// TIA Portal V17 export
// export: Created 2024-09-15T12:30:20.7468626Z, ExportSetting WithDefaults, DisplayName Totally Integrated Automation Portal, DisplayVersion V17, DisplayName TIA Portal Openness, DisplayVersion V17, DisplayName TIA Portal Version Control Interface, DisplayVersion V17, DisplayName STEP 7 Professional, DisplayVersion V17, DisplayName STEP 7 Safety, DisplayVersion V17, DisplayName WinCC Professional, DisplayVersion V17
VAR_GLOBAL   // PLC tag table "VGR - Vacuum Gripper Robot"
   IX_VGR_RefSwitchVerticalAxis_I1 AT %I1.6 : Bool;   // VGR - I1 = Reference switch vertical axis   {ExternalAccessible false, ExternalVisible false, ExternalWritable false}
   IX_VGR_RefSwitchHorizontalAxis_I2 AT %I3.6 : Bool;   // VGR - I2 = Reference switch horizontal axis   {ExternalAccessible false, ExternalVisible false, ExternalWritable false}
   IX_VGR_RefSwitchRotate_I3 AT %I3.7 : Bool;   // VGR - I3 = Reference switch rotate   {ExternalAccessible false, ExternalVisible false, ExternalWritable false}
   IX_VGR_EncoderVerticalAxisImp1_B1 AT %I6.0 : Bool;   // VGR - B1 = Encoder vertical axis imulse 1   {ExternalAccessible false, ExternalVisible false, ExternalWritable false}
   IX_VGR_EncoderVerticalAxisImp2_B2 AT %I6.4 : Bool;   // VGR - B2 = Encoder vertical axis imulse 2   {ExternalAccessible false, ExternalVisible false, ExternalWritable false}
   IX_VGR_EncoderHorizontalAxisImp1_B3 AT %I6.1 : Bool;   // VGR - B3 = Encoder horizontal axis imulse 1   {ExternalAccessible false, ExternalVisible false, ExternalWritable false}
   IX_VGR_EncoderHorizontalAxisImp2_B4 AT %I6.5 : Bool;   // VGR - B4 = Encoder horizontal axis imulse 2   {ExternalAccessible false, ExternalVisible false, ExternalWritable false}
   IX_VGR_EncoderRotateImp1_B5 AT %I6.2 : Bool;   // VGR - B5 = Encoder rotate impulse 1   {ExternalAccessible false, ExternalVisible false, ExternalWritable false}
   IX_VGR_EncoderRotateImp2_B6 AT %I6.6 : Bool;   // VGR - B6 = Encoder rotate impulse 2   {ExternalAccessible false, ExternalVisible false, ExternalWritable false}
   QX_VGR_M1_VerticalAxisUp_Q1 AT %Q2.0 : Bool;   // VGR - Q1 = Motor M1 vertical axis up   {ExternalAccessible false, ExternalVisible false, ExternalWritable false}
   QX_VGR_M1_VerticalAxisDown_Q2 AT %Q2.1 : Bool;   // VGR - Q2 = Motor M1 vertical axis down   {ExternalAccessible false, ExternalVisible false, ExternalWritable false}
   QX_VGR_M2_HorizontalAxisBackward_Q3 AT %Q2.2 : Bool;   // VGR - Q3 = Motor M2 horizontal axis backward   {ExternalAccessible false, ExternalVisible false, ExternalWritable false}
   QX_VGR_M2_HorizontalAxisForward_Q4 AT %Q2.3 : Bool;   // VGR - Q4 = Motor M2 horizontal axis forward   {ExternalAccessible false, ExternalVisible false, ExternalWritable false}
   QX_VGR_M3_RotateClockwise_Q5 AT %Q2.4 : Bool;   // VGR - Q5 = Motor M3 rotate clockwise   {ExternalAccessible false, ExternalVisible false, ExternalWritable false}
   QX_VGR_M3_RotateCounterclockwise_Q6 AT %Q2.5 : Bool;   // VGR - Q6 = Motor M3 rotate counterclockwise   {ExternalAccessible false, ExternalVisible false, ExternalWritable false}
   QX_VGR_Compressor_Q7 AT %Q2.6 : Bool;   // VGR - Q7 = Compressor   {ExternalAccessible false, ExternalVisible false, ExternalWritable false}
   QX_VGR_ValveVacuum_Q8 AT %Q2.7 : Bool;   // VGR - Q8 = Valve vacuum   {ExternalAccessible false, ExternalVisible false, ExternalWritable false}
   QW_VGR_PWM_Vertical_M1 AT %QW15 : Int;   // VGR = PWM Motor M1 vertical axis   {ExternalAccessible false, ExternalVisible false, ExternalWritable false}
   QW_VGR_PWM_Horizontal_M2 AT %QW17 : Int;   // VGR = PWM Motor M2 horizontal axis   {ExternalAccessible false, ExternalVisible false, ExternalWritable false}
   QW_VGR_PWM_Rotate_M3 AT %QW19 : Int;   // VGR = PWM Motor M3 rotate axis   {ExternalAccessible false, ExternalVisible false, ExternalWritable false}
END_VAR
